Staubli VAL3: __ts_german.pgx

program __ts_german()
begin
  //
end
